(* CODESYS project RESTAURANTE.project

Project tree, tasks and I/O mapping:
  Device : CODESYS Control Win V3, 3S - Smart Software Solutions GmbH, order no. 305021, version 3.5.11.30
    application Application
      libraries: Standard, * (System)
      task MainTask (cyclic, interval t#20ms, priority 1) calls PLC_PRG
      program PLC_PRG [LD]
*)

// Device/Application/PLC_PRG
PROGRAM PLC_PRG
VAR
	B1 : BOOL;
	ABERTO : BOOL;
	S1 : BOOL;
	S2 : BOOL;
	RESET : BOOL;
	PESSOAS : INT;
	VAZIO : BOOL;
	FECHADO: BOOL;
	CTUD_1: CTUD;
	LOTADO: BOOL;
END_VAR

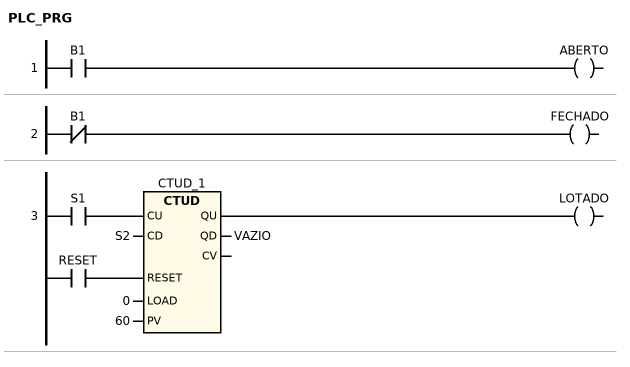
// NETWORK 1
ABERTO := B1;

// NETWORK 2
FECHADO := NOT B1;

// NETWORK 3
CTUD_1(CU := S1, CD := S2, RESET := RESET, LOAD := 0, PV := 60, QD => VAZIO); // CTUD
LOTADO := CTUD_1.QU;

END_PROGRAM
